// TIA Portal V19 export
DATA_BLOCK "Unit3Parameters"   // DB108
// stored: InstanceOfName LAF_typeHmiNgSortlUnitParameters, InstanceOfType UDT
"LAF_typeHmiNgSortlUnitParameters"
   // VAR
   //    em1 : "LAF_typeNgConveyorEm1ParametersHmi";
   // END_VAR
BEGIN
END_DATA_BLOCK
